{attribute 'qualified_only'}
{attribute 'strict'}
TYPE E_Message_BatteryInverter :
(
	eNoMessage := 0,
	eTooMuchBatteryInverter := 1,
	eBatteryInverterError := 2,
	eNoConnectionToBackend := 3
);
END_TYPE

(* stored: Version 1.1.0.1, ProductVersion 3.1.4024.6
   DUT E_Message_BatteryInverter: Id {d58dc19c-6fc6-4eed-bc1c-cef58ed16529} *)
